{attribute 'GeneratedUsingTerminal: KL8548'}
{attribute addProperty BoxType "KL8548"}
{attribute addProperty Id "Channel_1AT %Q*Channel_6576A6810Channel_2AT %Q*Channel_6576A6810Channel_3AT %Q*Channel_6576A6810Channel_4AT %Q*Channel_6576A6810Channel_5AT %Q*Channel_6576A6810Channel_6AT %Q*Channel_6576A6810Channel_7AT %Q*Channel_6576A6810Channel_8AT %Q*Channel_6576A6810"}
{attribute addProperty CRC "591730472"}
{attribute addProperty Size "0"}
TYPE KL8548_23451728 :
STRUCT
	{attribute addProperty Name "Channel_1"}
	Channel_1 : Channel_6576A681;
	{attribute addProperty Name "Channel_2"}
	Channel_2 : Channel_6576A681;
	{attribute addProperty Name "Channel_3"}
	Channel_3 : Channel_6576A681;
	{attribute addProperty Name "Channel_4"}
	Channel_4 : Channel_6576A681;
	{attribute addProperty Name "Channel_5"}
	Channel_5 : Channel_6576A681;
	{attribute addProperty Name "Channel_6"}
	Channel_6 : Channel_6576A681;
	{attribute addProperty Name "Channel_7"}
	Channel_7 : Channel_6576A681;
	{attribute addProperty Name "Channel_8"}
	Channel_8 : Channel_6576A681;
END_STRUCT
END_TYPE

(* stored: Version 1.2.0.0, ProductVersion 3.1.4024.9
   DUT KL8548_23451728: Id {b3fdd02f-2ec1-44d0-8e85-62baa43325d4} *)
